Fanuc KAREL source: kb00190.KL

-- PROVISIONAL review KL for V770-1; original PC SHA256 538e4e102b5c4dbcc01a4f9666e6d83e252fd924465f6779b3f329984f4f2c83
-- Incomplete behavior may be omitted. Consult companion uncertainty JSON. Do not deploy.
PROGRAM KB00190
%NOLOCKGROUP
VAR
  P1 : REAL
  RESULT : REAL
BEGIN
  -- UNRESOLVED_PC offsets 5-16; opcodes 2E,23
  -- UNRESOLVED_PC offsets 21-36; opcodes 27,22,76,23
  -- UNRESOLVED_PC offsets 41-45; opcodes 7F
END KB00190
